ABB RobotStudio station: Alushi_Yumi_EGM_2024.rspag

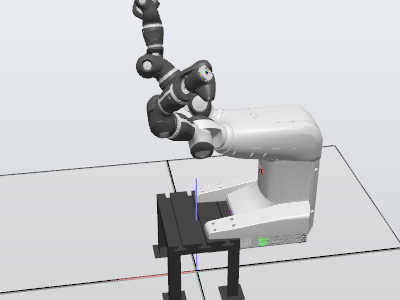
--- station ---
Station Alushi_Yumi_EGM_2024 (saved by RobotStudio 23.2.10395.0)
Controller YuMi_EGM_Alushi_2024, task T_ROB_L: task frame (RAPID world) sits at (-150, 0, 308) mm in the station
Controller YuMi_EGM_Alushi_2024, task T_ROB_R: task frame (RAPID world) sits at (-150, 0, 308) mm in the station
Controller YuMi_EGM_Alushi_2024
  mechanical unit ROB_R: IRB14000_0.5_0.5_R, 6 joints, base frame (0, 0, 0) mm
  mechanical unit ROB_R_7: IRB14000_0.5_0.5_R, 1 joints, base frame (0, 0, 0) mm
  mechanical unit ROB_L: IRB14000_0.5_0.5_L, 6 joints, base frame (0, 0, 0) mm
  mechanical unit ROB_L_7: IRB14000_0.5_0.5_L, 1 joints, base frame (0, 0, 0) mm
Layout (positions relative to the parent item):
  - table [part] at (175, -225, 0) mm, rotated rx 0 ry 0 rz 90 deg, size 450 x 350 x 308 mm
  - IRB14000_0.5_0.5 [mechanism, from %ABB.RobotStudio.Models.IRB14000%\IRB14000_0.5_0.5__02.rslib] at (-150, 0, 308) mm
  - IRB14000_0.5_0.5_R [mechanism, from %ABB.RobotStudio.Models.IRB14000%\IRB14000_0.5_0.5__02.rslib] at (-150, 0, 308) mm; joint values [-0.3598, -0.3596, -0.0003, -2.1255, 0, -0.5344, 0] (rad or m)
  - IRB14000_0.5_0.5_L [mechanism, from %ABB.RobotStudio.Models.IRB14000%\IRB14000_0.5_0.5__02.rslib] at (-150, 0, 308) mm; joint values [-2.903, -0.0009, -0.0003, -0.0002, 0, -0.0001, 0] (rad or m)

--- Controller Data/YuMi_EGM_Alushi_2024/RAPID/TASK1/PROGMOD/Module_Right_Arm_IRB14000.mod ---
MODULE Module_Right_Arm_IRB14000
    !***********************************************************
    !
    ! Module     :  Module_Right_Arm_IRB14000
    ! Description:
    !   ABB YuMi IRB1400 Right Arm Module for Externally Guided Motion [EGM]
    !   using UdpUc external sensor - setup for communication over
    !   Robot Operating System (ROS)
    ! Author     : Alushi
    ! Supervisor : K.Al Khudir
    ! Version    : 1.0
    ! Date       : 06/2024
    !***********************************************************

    !***********************************************************
    ! Procedure main
    !   This is the program entry point
    !***********************************************************

VAR egmident channel_2;
    VAR egmstate egmSt2;
    ! Adjust these constants to the limits that make sense for your application.
    CONST egm_minmax egm_minmax_lin1:=[-1,1]; ! in mm
    CONST egm_minmax egm_minmax_rot1:=[-2,2]; ! in degrees
    CONST egm_minmax egm_minmax_joint1:=[-0.5,0.5]; ! in radians or degrees based on your system setup

  PROC main()
        VAR jointtarget joints;
        ! "Move" a tiny amount to start EGM; externally guided motion may only begin from fine point.
        joints:= CJointT();                   ! Reads current joint angles for move to current pose
        MoveAbsj joints, v1000, fine, tool0;  ! Ensure velocity and zone data are appropriate for your robot.
        StartEGM;
        ! Start EGM action here:
        EGMActJoint channel_2 \Tool:=tool0 \WObj:=wobj0, \J1:=egm_minmax_joint1 \J2:=egm_minmax_joint1 \J3:=egm_minmax_joint1
        \J4:=egm_minmax_joint1 \J5:=egm_minmax_joint1 \J6:=egm_minmax_joint1 \J7:=egm_minmax_joint1 \LpFilter:=100 \Samplerate:=4 \MaxPosDeviation:=1000 \MaxSpeedDeviation:=10000;
        ! Start the EGM joint movement.
        EGMRunJoint channel_2, EGM_STOP_HOLD \J1 \J2 \J3 \J4 \J5 \J6 \J7 \CondTime:=2000000 \RampInTime:=0.01 \PosCorrGain:=0;
        ! An infinite loop to keep the robot running in EGM
        WHILE TRUE DO
            WaitTime 1;                       ! Adjustable for suitable cycle time for application.
        ENDWHILE
        ExitCycle;                            ! Exit the procedure on error or interruption.
    ERROR
        TPWrite "An error occurred.";         ! Handle errors as appropriate for your application.
        RAISE;
    ENDPROC

    PROC StartEGM()
        EGMGetId channel_2;                   ! Obtain a unique EGM identifier.
        egmSt2 := EGMGetState(channel_2);
        IF egmSt2 <= EGM_STATE_CONNECTED THEN ! Set up EGM if the robot is not yet connected.
            EGMSetupUC ROB_R, channel_2, "ConfR", "UCdeviceR:" \Joint \CommTimeout:=10000;
        ENDIF
        EGMStreamStart channel_2;             ! Start EGM stream.
    ENDPROC

ENDMODULE

--- Controller Data/YuMi_EGM_Alushi_2024/RAPID/TASK2/PROGMOD/Module_Left_Arm_IRB14000.mod ---
MODULE Module_Left_Arm_IRB14000
    !***********************************************************
    !
    ! Module     :  Module_Left_Arm_IRB14000
    ! Description:
    !   ABB YuMi IRB14000 Left Arm Module for Externally Guided Motion [EGM]
    !   using UdpUc external sensor - setup for communication over
    !   Robot Operating System (ROS)
    ! Author     : Alushi
    ! Supervisor : K.Al Khudir
    ! Version    : 1.0
    !
    !***********************************************************

    !***********************************************************
    ! Procedure main
    !   This is the program entry point
    !***********************************************************

VAR egmident channel_1;
    VAR egmstate egmSt1;
    ! Adjust these constants to the limits that make sense for your application.
    CONST egm_minmax egm_minmax_lin1:=[-1,1]; ! in mm
    CONST egm_minmax egm_minmax_rot1:=[-2,2]; ! in degrees
    CONST egm_minmax egm_minmax_joint1:=[-0.5,0.5]; ! in radians or degrees based on your system setup

  PROC main()
        VAR jointtarget joints;
        ! "Move" a tiny amount to start EGM; externally guided motion may only begin from fine point.
        joints:= CJointT();                   ! Reads current joint angles for move to current pose
        MoveAbsj joints, v1000, fine, tool0;  ! Ensure velocity and zone data are appropriate for your robot.
        StartEGM;
        ! Start EGM action here:
        EGMActJoint channel_1 \Tool:=tool0 \WObj:=wobj0, \J1:=egm_minmax_joint1 \J2:=egm_minmax_joint1 \J3:=egm_minmax_joint1
        \J4:=egm_minmax_joint1 \J5:=egm_minmax_joint1 \J6:=egm_minmax_joint1 \J7:=egm_minmax_joint1 \LpFilter:=100 \Samplerate:=4 \MaxPosDeviation:=1000 \MaxSpeedDeviation:=10000;
        ! Start the EGM joint movement.
        EGMRunJoint channel_1, EGM_STOP_HOLD \J1 \J2 \J3 \J4 \J5 \J6 \J7 \CondTime:=2000000 \RampInTime:=0.01 \PosCorrGain:=0;
        ! An infinite loop to keep the robot running in EGM
        WHILE TRUE DO
            WaitTime 1;                       ! Adjustable for suitable cycle time for application.
        ENDWHILE
        ExitCycle;                            ! Exit the procedure on error or interruption.
    ERROR
        TPWrite "An error occurred.";         ! Handle errors as appropriate for your application.
        RAISE;
    ENDPROC

    PROC StartEGM()
        EGMGetId channel_1;                   ! Obtain a unique EGM identifier.
        egmSt1 := EGMGetState(channel_1);
        IF egmSt1 <= EGM_STATE_CONNECTED THEN ! Set up EGM if the robot is not yet connected.
            EGMSetupUC ROB_L, channel_1, "ConfL", "UCdeviceL:" \Joint \CommTimeout:=10000;
        ENDIF
        EGMStreamStart channel_1;             ! Start EGM stream.
    ENDPROC

ENDMODULE

--- Controller Data/YuMi_EGM_Alushi_2024/SYSPAR/EIO.cfg ---
EIO:CFG_1.0:6:1::
#
SYSSIG_IN:

      -Signal "Collision_Avoidance" -Action "CollAvoidance"
#
INDUSTRIAL_NETWORK:

      -Name "EtherNetIP" -Connection "Private Network"\
      -Label "EtherNet/IP Adapter Network"

      -Name "DeviceNet" -Label "DeviceNet Master/Slave Network" -Address "2"
#
EIO_CROSS:

      -Name "Cross_Signal_Lamp" -Res "Signal_Lamp" -Act1 "DRV1BRAKE"
#
EIO_SIGNAL_SAFELEVEL:

      -Name "FlangePowerSafeLevel" -ActionWhenStartup "Last"
#
DEVICENET_DEVICE:

      -Name "D652_10" -VendorName "ABB Robotics" -ProductName "24 VDC Unit"\
      -Address 10 -ProductCode 26 -DeviceType 7 -ConnectionType "COS"\
      -OutputSize 2 -InputSize 2
#
DEVICENET_INTERNAL_DEVICE:

      -Name "DN_Internal_Device" -VendorName "ABB Robotics"\
      -ProductName "DeviceNet Internal Slave Device"
#
ETHERNETIP_INTERNAL_DEVICE:

      -Name "EN_Internal_Device" -VendorName "ABB Robotics"\
      -ProductName "EtherNet/IP Internal Adapter Device"
#
EIO_SIGNAL:

      -Name "custom_DI_0" -SignalType "DI" -Device "D652_10" -DeviceMap "0"

      -Name "custom_DI_1" -SignalType "DI" -Device "D652_10" -DeviceMap "1"

      -Name "custom_DI_2" -SignalType "DI" -Device "D652_10" -DeviceMap "2"

      -Name "custom_DI_3" -SignalType "DI" -Device "D652_10" -DeviceMap "3"

      -Name "custom_DI_4" -SignalType "DI" -Device "D652_10" -DeviceMap "4"

      -Name "custom_DI_5" -SignalType "DI" -Device "D652_10" -DeviceMap "5"

      -Name "custom_DI_6" -SignalType "DI" -Device "D652_10" -DeviceMap "6"

      -Name "custom_DI_7" -SignalType "DI" -Device "D652_10" -DeviceMap "7"

      -Name "custom_DO_0" -SignalType "DO" -Device "D652_10" -DeviceMap "0"

      -Name "custom_DO_1" -SignalType "DO" -Device "D652_10" -DeviceMap "1"

      -Name "custom_DO_2" -SignalType "DO" -Device "D652_10" -DeviceMap "2"

      -Name "custom_DO_3" -SignalType "DO" -Device "D652_10" -DeviceMap "3"

      -Name "custom_DO_4" -SignalType "DO" -Device "D652_10" -DeviceMap "4"

      -Name "custom_DO_5" -SignalType "DO" -Device "D652_10" -DeviceMap "5"

      -Name "custom_DO_6" -SignalType "DO" -Device "D652_10" -DeviceMap "6"

      -Name "custom_DO_7" -SignalType "DO" -Device "D652_10" -DeviceMap "7"

      -Name "hall_sensor_joint_1" -SignalType "DI" -Device "D652_10"\
      -DeviceMap "8"

      -Name "hall_sensor_joint_2" -SignalType "DI" -Device "D652_10"\
      -DeviceMap "9"

      -Name "hall_sensor_joint_3" -SignalType "DI" -Device "D652_10"\
      -DeviceMap "11"

      -Name "hall_sensor_joint_4" -SignalType "DI" -Device "D652_10"\
      -DeviceMap "12"

      -Name "hall_sensor_joint_5" -SignalType "DI" -Device "D652_10"\
      -DeviceMap "13"

      -Name "hall_sensor_joint_6" -SignalType "DI" -Device "D652_10"\
      -DeviceMap "14"

      -Name "hall_sensor_joint_7" -SignalType "DI" -Device "D652_10"\
      -DeviceMap "10"

      -Name "hall_sensor_24V_ROB_R" -SignalType "DO" -Device "D652_10"\
      -DeviceMap "8"

      -Name "hall_sensor_24V_ROB_L" -SignalType "DO" -Device "D652_10"\
      -DeviceMap "9"

      -Name "flange_24V_ROB_R" -SignalType "DO" -Device "D652_10"\
      -DeviceMap "10" -SafeLevel "FlangePowerSafeLevel"

      -Name "flange_24V_ROB_L" -SignalType "DO" -Device "D652_10"\
      -DeviceMap "11" -SafeLevel "FlangePowerSafeLevel"

      -Name "Signal_Lamp" -SignalType "DO" -Device "D652_10" -DeviceMap "12"

      -Name "Collision_Avoidance" -SignalType "DO" -Access "All" -Default 1
